// TIA Portal V16 export
// export: Created 2021-05-25T16:14:40.0390091Z, ExportSetting WithDefaults, DisplayName Totally Integrated Automation Portal, DisplayVersion V16, DisplayName TIA Portal Version Control Interface, DisplayVersion V16, DisplayName TIA Portal Openness, DisplayVersion V16, DisplayName STEP 7 Professional, DisplayVersion V16, DisplayName STEP 7 Safety, DisplayVersion V16, DisplayName WinCC Unified SCADA Engineering System, DisplayVersion V16
DATA_BLOCK "dbDigitalSensors"   // DB30
{ S7_Optimized_Access := 'FALSE'; DB_Accessible_From_OPC_UA := 'FALSE' }
VERSION : 0.1
// stored: AutoNumber false, DBAccessibleFromOPCUA false, IsOnlyStoredInLoadMemory false, IsWriteProtectedInAS false
   VAR
      ZAUSTAVITEV_V_SILI_NI_AKTIVIRANA : "udtDigitalSensor";
      FOTO_ZAVESA_KANAL_1 : "udtDigitalSensor";
      FOTO_ZAVESA_KANAL_2 : "udtDigitalSensor";
      START_LEVO_NA_VPENJANJU : "udtDigitalSensor";
      START_DESNO_NA_VPENJANJU : "udtDigitalSensor";
      PRISOTNOST_ZRAKA_NA_NAPRAVI : "udtDigitalSensor";
      BIMETAL_TRANSPORTA_NOGIC_IZKLJUCIL : "udtDigitalSensor";
      VIBRATOR_NOGIC_READY : "udtDigitalSensor";
      BIMETAL_VIJACENJA_NOGIC_IZKLJUCIL : "udtDigitalSensor";
      FR_MOTORJA1_ZADAJ_DESNO_READY : "udtDigitalSensor";
      FR_MOTORJA2_SPREDAJ_DESNO_READY : "udtDigitalSensor";
      FR_MOTORJA1_ZADAJ_LEVO_READY : "udtDigitalSensor";
      FR_MOTORJA2_SPREDAJ_LEVO_READY : "udtDigitalSensor";
      Spare20_7 : "udtDigitalSensor";
      FOTOCELICA_TRANSPORTA_NOGIC : "udtDigitalSensor";
      FOTOCELICA_VSTOP_DRCA_NOGIC : "udtDigitalSensor";
      FOTOCELICA_PRED_MESTOM_LOCEVANJA : "udtDigitalSensor";
      FOTOCELICA_VSTOP_DRCA_LEVO : "udtDigitalSensor";
      FOTOCELICA_VSTOP_DRCA_DESNO : "udtDigitalSensor";
      FOTOCELICA_LOC_IZH_DRCA_LEVO : "udtDigitalSensor";
      FOTOCELICA_LOC_IZH_DRCA_DESNO : "udtDigitalSensor";
      NOGICE_V_VIBRATORJU : "udtDigitalSensor";
      ROTACIJSKI_CIL_DESNO : "udtDigitalSensor";
      ROTACIJSKI_CIL_SREDINA : "udtDigitalSensor";
      ROTACIJSKI_CIL_LEVO : "udtDigitalSensor";
      LOC_DRCA_DESNO_NAPREJ : "udtDigitalSensor";
      LOC_DRCA_DESNO_NAZAJ : "udtDigitalSensor";
      LOC_DRCA_LEVO_NAZAJ : "udtDigitalSensor";
      LOC_DRCA_LEVO_NAPREJ : "udtDigitalSensor";
      Spare22_7 : "udtDigitalSensor";
      FOTOCELICA_LOC_TRAK_DESNO1 : "udtDigitalSensor";
      FOTOCELICA_LOC_TRAK_DESNO2 : "udtDigitalSensor";
      FOTOCELICA_VIJACENJE_DESNOZADAJ : "udtDigitalSensor";
      FOTOCELICA_VIJACENJE_DESNOSPREDAJ : "udtDigitalSensor";
      VIJACENJE_DESNO_1_NAZAJ : "udtDigitalSensor";
      VIJACENJE_DESNO_1_NAPREJ : "udtDigitalSensor";
      MESTO_VIJAC_STOP_DESNO_ZAD_NAZAJ : "udtDigitalSensor";
      MESTO_VIJAC_STOP_DESNO_ZAD_NAPREJ : "udtDigitalSensor";
      MESTO_VIJACENJE_DESNO_ZAD_DVIG_DOL : "udtDigitalSensor";
      MESTO_VIJACENJE_DESNO_ZAD_CENT_NARAZEN : "udtDigitalSensor";
      MESTO_VIJACENJE_DESNO_ZAD_CENT_SKUPAJ : "udtDigitalSensor";
      Spare24_3 : "udtDigitalSensor";
      Spare24_4 : "udtDigitalSensor";
      MESTO_VIJACENJE_DESNO_SPRED_DVIG_DOL : "udtDigitalSensor";
      MESTO_VIJACENJE_DESNO_SPRED_CENT_NARAZEN : "udtDigitalSensor";
      MESTO_VIJACENJE_DESNO_SPRED_CENT_SKUPAJ : "udtDigitalSensor";
      KONCNA_POZICIJA_VIJACENJA_DES_NAZAJ : "udtDigitalSensor";
      KONCNA_POZICIJA_VIJACENJA_DES_NAPREJ : "udtDigitalSensor";
      Spare25_2 : "udtDigitalSensor";
      Spare25_3 : "udtDigitalSensor";
      KONCNA_POZICIJA_VIJACENJA_LEVO_NAZAJ : "udtDigitalSensor";
      KONCNA_POZICIJA_VIJACENJA_LEVO_NAPREJ : "udtDigitalSensor";
      Spare25_6 : "udtDigitalSensor";
      Spare25_7 : "udtDigitalSensor";
      FOTOCELICA_LOC_TRAK_LEVO1 : "udtDigitalSensor";
      FOTOCELICA_LOC_TRAK_LEVO2 : "udtDigitalSensor";
      FOTOCELICA_VIJACENJE_LEVO_ZADAJ : "udtDigitalSensor";
      FOTOCELICA_VIJACENJE_LEVO_SPREDAJ : "udtDigitalSensor";
      VIJACENJE_LEVO_1_NAZAJ : "udtDigitalSensor";
      VIJACENJE_LEVO_1_NAPREJ : "udtDigitalSensor";
      MESTO_VIJAC_STOP_LEVO_ZAD_NAZAJ : "udtDigitalSensor";
      MESTO_VIJAC_STOP_LEVO_ZAD_NAPREJ : "udtDigitalSensor";
      MESTO_VIJACENJE_LEVO_ZAD_DVIG_DOL : "udtDigitalSensor";
      MESTO_VIJACENJE_LEVO_ZAD_CENT_NARAZEN : "udtDigitalSensor";
      MESTO_VIJACENJE_LEVO_ZAD_CENT_SKUPAJ : "udtDigitalSensor";
      Spare27_3 : "udtDigitalSensor";
      Spare27_4 : "udtDigitalSensor";
      MESTO_VIJACENJE_LEVO_SPRED_DVIG_DOL : "udtDigitalSensor";
      MESTO_VIJACENJE_LEVO_SPRED_CENT_NARAZEN : "udtDigitalSensor";
      MESTO_VIJACENJE_LEVO_SPRED_CENT_SKUPAJ : "udtDigitalSensor";
      INDUKTIVEC_PRAVILNA_VLOZITEV_DNA_1 : "udtDigitalSensor";
      INDUKTIVEC_PRAVILNA_VLOZITEV_DNA_2 : "udtDigitalSensor";
      VPENJANJE_DNA_LEVO_ZADAJ_GOR : "udtDigitalSensor";
      VPENJANJE_DNA_LEVO_ZADAJ_DOL : "udtDigitalSensor";
      VPENJANJE_DNA_LEVO_SPREDAJ_GOR : "udtDigitalSensor";
      VPENJANJE_DNA_LEVO_SPREDAJ_DOL : "udtDigitalSensor";
      VPENJANJE_DNA_DESNO_ZADAJ_GOR : "udtDigitalSensor";
      VPENJANJE_DNA_DESNO_ZADAJ_DOL : "udtDigitalSensor";
      VPENJANJE_DNA_DESNO_SPREDAJ_GOR : "udtDigitalSensor";
      VPENJANJE_DNA_DESNO_SPREDAJ_DOL : "udtDigitalSensor";
   END_VAR
BEGIN
END_DATA_BLOCK
